PROGRAM WORLD_WEATHER_DEMO
VAR
	IP_C: IP_C;
	S_BUF: NETWORK_BUFFER;
	R_BUF: NETWORK_BUFFER;
	IP_CONTROL_1: IP_CONTROL;
	activate: BOOL := TRUE;
	done: BOOL;
	busy: BOOL;
	error_c: DWORD;
	error_t: BYTE;
	latitude: REAL := 48.21;
	longitude: REAL := 16.37;
	WORLD_WEATHER: WORLD_WEATHER;
	WW_DATA: WORLD_WEATHER_DATA;
	CLK_PRG: CLK_PRG;
	WORLD_WEATHER_DESC_GE: WORLD_WEATHER_DESC_GE;
	WORLD_WEATHER_ICON_OSCAT: WORLD_WEATHER_ICON_OSCAT;
END_VAR
VAR // added by the converter: edge detectors and wires of the graphical bodies
    _w1 : ANY;
END_VAR

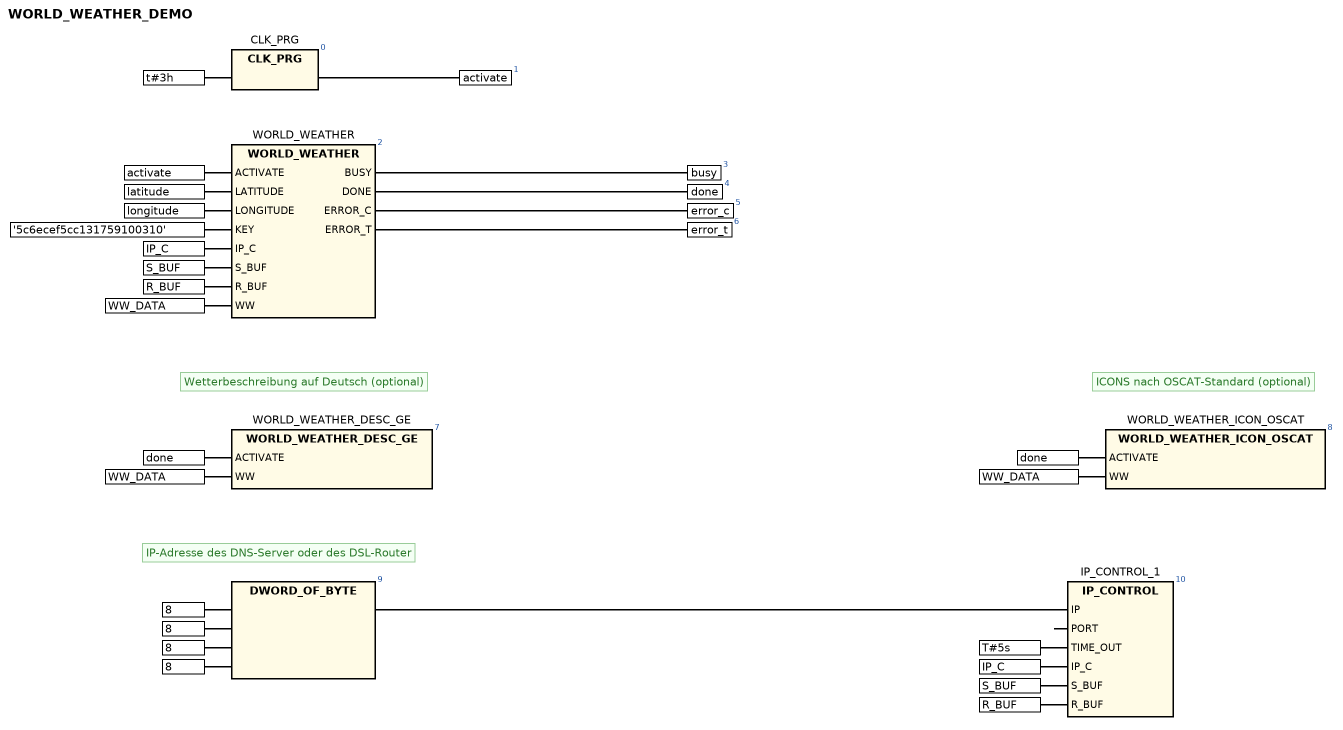
CLK_PRG(_in1 := t#3h);
activate := CLK_PRG._out1;
WORLD_WEATHER(
    ACTIVATE := activate,
    LATITUDE := latitude,
    LONGITUDE := longitude,
    KEY := '5c6ecef5cc131759100310',
    IP_C := IP_C,
    S_BUF := S_BUF,
    R_BUF := R_BUF,
    WW := WW_DATA);
busy := WORLD_WEATHER.BUSY;
done := WORLD_WEATHER.DONE;
error_c := WORLD_WEATHER.ERROR_C;
error_t := WORLD_WEATHER.ERROR_T;
// Wetterbeschreibung auf Deutsch (optional)
WORLD_WEATHER_DESC_GE(ACTIVATE := done, WW := WW_DATA);
// ICONS nach OSCAT-Standard (optional)
WORLD_WEATHER_ICON_OSCAT(ACTIVATE := done, WW := WW_DATA);
// IP-Adresse des DNS-Server oder des DSL-Router
_w1 := DWORD_OF_BYTE(8, 8, 8, 8);
IP_CONTROL_1(IP := _w1, TIME_OUT := T#5s, IP_C := IP_C, S_BUF := S_BUF, R_BUF := R_BUF); // IP_CONTROL

END_PROGRAM

(* stored: Version 1.1.0.1, ProductVersion 3.1.4022.7
   POU WORLD_WEATHER_DEMO: Id {e24bf8a9-31da-46ef-9376-70d71bbd1193}, SpecialFunc None *)
